(* Schneider Machine Expert - Basic project SCALLING BLOCK UDFB, file version 2.7.0.0 *)
(* ProjectInformations: Name=New project *)

HARDWARE
  Cpu 0: TM221CE16U
  ModuleExtensionObject 0: TM3AM6/G
  EthernetConfiguration: NetworkName=M221, IpAllocationMode=FixedAddress, IpAddress=0.0.0.0, SubnetMask=0.0.0.0
  SerialLineConfiguration: Baud=Baud19200, Parity=ParityEven, DataBits=DataBits8, StopBits=StopBits1, PhysicalMedium=PhysicalMediumRs485, TransmissionMode=TransmissionModeModbusRtu, SlaveId=1, Addressing=SlaveAddressing
  MastTask: UsePeriodScanMode=false, PeriodScan=100
  FastTask: Period=255
  CpuBehavior: StartingMode=StartAsPreviousState, AutoSaveRamOnEeprom=true, WatchdogPeriod=250

SYMBOLS  (address, symbol, comment, settings)
  %S5       SB_TB100MS  "Time base of 100 ms generated by an internal clock"
  %MF100    AI_MIN
  %MF102    AI_MAX
  %MF104    SENSOR_MIN
  %MF106    SENSOR_MAX
  %MF108    ACTUAL

POU SCALLING
  (* SectionNumber=1 *)

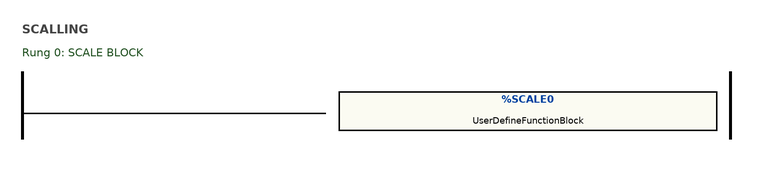

// Rung 0: SCALE BLOCK
  LD 1
  BLK_UDFB 2
  LD 1
  ST %UDF0.PARAMW9:X0
  LD 1
  ST %UDF0.PARAMW9:X8
  [ %UDF0.PARAMF0 := %SCALE0.RAW_VALUE_F ]
  [ %UDF0.PARAMF1 := %SCALE0.AI_MIN ]
  [ %UDF0.PARAMF2 := %SCALE0.AI_MAX ]
  [ %UDF0.PARAMF3 := %SCALE0.SENSOR_MIN ]
  [ %UDF0.PARAMF4 := %SCALE0.SENSOR_MAX ]
  [ %UDF0.PARAMF5 := %SCALE0.ACTUAL ]
  [ %UDF0.PARAMW6 := %SCALE0.RAW_VALUE_W ]
  [ %UDF0.PARAMF7 := %SCALE0.PARAM0 ]
  [ %UDF0.PARAMF8 := %SCALE0.PARAM1 ]
  [ %UDF0.RETW0 := %UDF1.RETW0 ]
  [ %UDF0.RETW1 := %UDF1.RETW1 ]
  [ %UDF0.RETW2 := %UDF1.RETW2 ]
  [ %UDF0.RETW3 := %UDF1.RETW3 ]
  UDF0
  [ %UDF1.RETW0 := %UDF0.RETW0 ]
  [ %UDF1.RETW1 := %UDF0.RETW1 ]
  [ %UDF1.RETW2 := %UDF0.RETW2 ]
  [ %UDF1.RETW3 := %UDF0.RETW3 ]
  [ %SCALE0.RAW_VALUE_F := %UDF0.PARAMF0 ]
  [ %SCALE0.AI_MIN := %UDF0.PARAMF1 ]
  [ %SCALE0.AI_MAX := %UDF0.PARAMF2 ]
  [ %SCALE0.SENSOR_MIN := %UDF0.PARAMF3 ]
  [ %SCALE0.SENSOR_MAX := %UDF0.PARAMF4 ]
  [ %SCALE0.ACTUAL := %UDF0.PARAMF5 ]
  [ %SCALE0.RAW_VALUE_W := %UDF0.PARAMW6 ]
  [ %SCALE0.PARAM0 := %UDF0.PARAMF7 ]
  [ %SCALE0.PARAM1 := %UDF0.PARAMF8 ]
  END_BLK_UDFB 2

POU SCALE DATA
  (* SectionNumber=2 *)

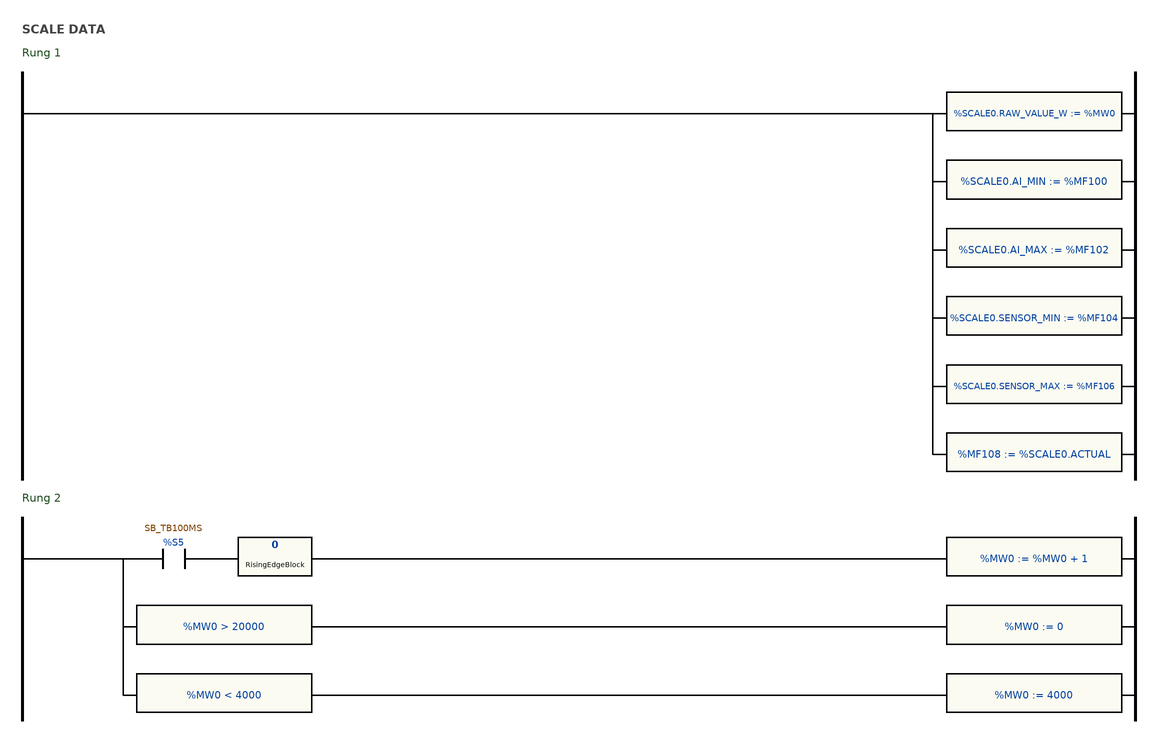

// Rung 1
  LD 1
  [ %SCALE0.RAW_VALUE_W := %MW0 ]
  [ %SCALE0.AI_MIN := %MF100 ](* AI_MIN *)
  [ %SCALE0.AI_MAX := %MF102 ](* AI_MAX *)
  [ %SCALE0.SENSOR_MIN := %MF104 ](* SENSOR_MIN *)
  [ %SCALE0.SENSOR_MAX := %MF106 ](* SENSOR_MAX *)
  [ %MF108 := %SCALE0.ACTUAL ](* ACTUAL *)
  // as ST:
  //   %SCALE0.RAW_VALUE_W := %MW0;
  //   %SCALE0.AI_MIN := AI_MIN;
  //   %SCALE0.AI_MAX := AI_MAX;
  //   %SCALE0.SENSOR_MIN := SENSOR_MIN;
  //   %SCALE0.SENSOR_MAX := SENSOR_MAX;
  //   ACTUAL := %SCALE0.ACTUAL;

// Rung 2
  LD 1
  MPS
  AND %S5                 (* SB_TB100MS *)
  RISING0
  [ %MW0 := %MW0 + 1 ]
  MRD
  AND [ %MW0 > 20000 ]
  [ %MW0 := 0 ]
  MPP
  AND [ %MW0 < 4000 ]
  [ %MW0 := 4000 ]
  // as ST:
  //   IF RISING(SB_TB100MS) THEN %MW0 := %MW0 + 1; END_IF;
  //   IF %MW0 > 20000 THEN %MW0 := 0; END_IF;
  //   IF %MW0 < 4000 THEN %MW0 := 4000; END_IF;

UserFunctionBlockPou SCALE
  (* SectionNumber=3 *)

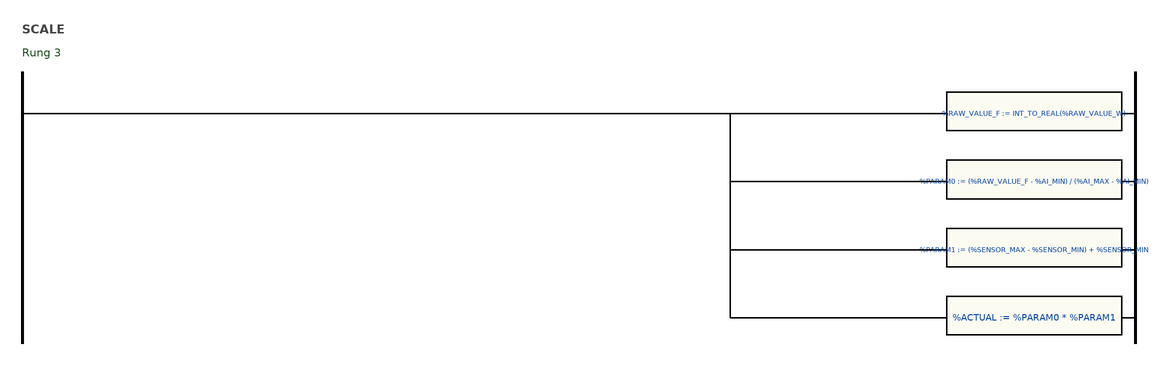

// Rung 3
  LD 1
  [ %RAW_VALUE_F := INT_TO_REAL ( %RAW_VALUE_W ) ]
  [ %PARAM0 := ( %RAW_VALUE_F - %AI_MIN ) / ( %AI_MAX - %AI_MIN ) ]
  [ %PARAM1 := ( %SENSOR_MAX - %SENSOR_MIN ) + %SENSOR_MIN ]
  [ %ACTUAL := %PARAM0 * %PARAM1 ]
  // as ST:
  //   %RAW_VALUE_F := INT_TO_REAL ( %RAW_VALUE_W );
  //   %PARAM0 := ( %RAW_VALUE_F - %AI_MIN ) / ( %AI_MAX - %AI_MIN );
  //   %PARAM1 := ( %SENSOR_MAX - %SENSOR_MIN ) + %SENSOR_MIN;
  //   %ACTUAL := %PARAM0 * %PARAM1;
